FUNCTION_BLOCK FB_CameraDummy EXTENDS FB_CameraBase
VAR_INPUT
END_VAR
VAR_OUTPUT
END_VAR
VAR
END_VAR

{attribute 'monitoring':='call'}
PROPERTY eCameraMode : E_CameraMode
GET
eCameraMode := _eCameraMode;
IF _eCameraMode = E_CameraMode.Auto THEN
  eCameraMode := E_CameraMode.NoCorrection;
END_IF
END_GET
END_PROPERTY

PROPERTY eDeviceType : E_CameraDevice
GET
eDeviceType := E_CameraDevice.SheetDetect;
END_GET
END_PROPERTY

METHOD GetCamStatus : BOOL
VAR_OUTPUT
  bConnectionOK  : BOOL;    // Camera connected
  bTeachOk       : BOOL;    // Teach successful
  nTeachedPoints : UDINT;   // Teached points for this job
  nScannedPoints : UDINT;   // Scanned points on current sheet
  bCamStarted    : BOOL;    // Camera trigger is active, cam started
  bCamDone       : BOOL;    // Camera finished on last CT
  bErrors        : ARRAY[1..GVL_Camera.nC_NbCamErrors] OF BOOL;  // generic error flag list
END_VAR
bConnectionOK  := TRUE;  //NO comm with a cam 
bTeachOk       := TRUE;  //NO teach availabe
nTeachedPoints := 0;
nScannedPoints := 0;
bCamStarted    := _bCamStarted;
bCamDone       := _bCamDone;

GetCamStatus := TRUE;
END_METHOD

(*
  Set mode to camera.
  :return: TRUE if success
*)
METHOD setCameraMode : BOOL
VAR_INPUT
  eCameraMode : E_CameraMode;
END_VAR
IF eCameraMode = E_CameraMode.NoCorrection THEN   // supported mode
  
  _eCameraMode := eCameraMode; 
  setCameraMode := TRUE;        // set desired mode
ELSE
  LogError(F_Concat3('Camera mode=', TO_STRING(eCameraMode), ' not supported by camera'));
  _eCameraMode := E_CameraMode.NoCorrection;
END_IF
END_METHOD

{attribute 'monitoring':='variable'}
PROPERTY sName : STRING
GET
sName := 'SheetDetect';
END_GET
END_PROPERTY

END_FUNCTION_BLOCK

(* stored: Version 1.1.0.1, ProductVersion 3.1.4024.3
   POU FB_CameraDummy: Id {25aa4386-39f0-469e-b501-cef0bb36b533}, SpecialFunc None
   Property eCameraMode: Id {6d0d2ebb-c8e7-4e49-b4bf-371007fb02f7}
   Get Get: Id {a84fecb9-d352-4caa-b5e8-ae26a7d3e977}
   Property eDeviceType: Id {6bc68d1d-d9b7-4b72-a72b-c1581c89809e}
   Get Get: Id {708013e7-3119-4cf9-8185-b1fc9c6336ee}
   Method GetCamStatus: Id {002a8acc-defe-4563-8b88-d149af9e57f9}
   Method setCameraMode: Id {e977affa-219b-4b8e-97d6-f357fdc03577}
   Property sName: Id {2f5c4c3d-a6df-4ad3-9917-b6a5986d4c5b}
   Get Get: Id {4445f55b-fc81-490f-b8b1-8b169e893684} *)
